Staubli VAL3: getObjectLatch.pgx

public program getObjectLatch(num x_nIdx (dimensions=1), num& x_nLatchedVal[] (dimensions=1))
begin
  // This program returns the latched encoder value of the detected object.
  //  This is useful only when the latched encoder value is given by the
  //  detection library and not by the encoder library, like in the case
  //  of the detection library "Socket".
  //
  // Input param
  //    x_nIdx         : Position of the object in the queue.
  //
  // Output param
  //    nObjectLatch   : Latched encoder value read from a socket.
  //
  //
  //----------------------------------------------------------------
  //
  x_nLatchedVal=nLatchedValue[x_nIdx]
  //
end
